Fanuc KAREL source: kc00049.KL

-- PROVISIONAL review KL for V940-1; original PC SHA256 bc40aea5b251ee67b8d016c4226a58f8446d2ee0afeef851056f46c2ca05c5c6
-- Incomplete behavior may be omitted. Consult companion uncertainty JSON. Do not deploy.
PROGRAM KC00049
%NOLOCKGROUP
BEGIN
  -- V9_ZERO_TABLE_METADATA_HINT layout=0002_ascii; no indexed target words; source/name/runtime held
  -- UNRESOLVED_PC offsets 5-35; opcodes 27,22,22,1C,22,27,9D,31
  -- UNRESOLVED_PC offsets 40-44; opcodes 7F
END KC00049
